FUNCTION_BLOCK PUBLIC FB_LampSetDirectDALI
VAR
	nLightLevel			: USINT;
	_nOperatingTime		: DINT;
	tonDelay			: TON;
END_VAR

IF (nLightLevel > 0) THEN
	tonDelay(IN := TRUE, PT := T#1S);
	IF (tonDelay.Q) THEN
		tonDelay(IN := FALSE);
		_nOperatingTime := _nOperatingTime + 1;
	END_IF
ELSE
	tonDelay(IN := FALSE);
END_IF

{attribute 'monitoring' := 'call'}
// Operating Time [s]
PROPERTY PUBLIC nOperatingTime : DINT
GET
nOperatingTime := _nOperatingTime;
END_GET
SET
_nOperatingTime := nOperatingTime;
END_SET
END_PROPERTY

// Sets the control value of the DALI lamp to a value between 0 and 254.
METHOD PUBLIC SetLightLevel
VAR_INPUT
	nNewLightLevel		: USINT(0..254);
END_VAR
nLightLevel := nNewLightLevel;
END_METHOD

END_FUNCTION_BLOCK

(* stored: Version 1.1.0.1, ProductVersion 3.1.4024.12
   POU FB_LampSetDirectDALI: Id {508b93c0-0778-4ff1-aedf-858d8647b6a3}, SpecialFunc None
   Property nOperatingTime: Id {62d392a4-ac0b-46a0-b328-e579ec751c57}
   Get Get: Id {329a3336-a875-4ed5-8e94-b64093512612}
   Set Set: Id {193ef73e-2d46-4bd6-be4a-aedf24d1322f}
   Method SetLightLevel: Id {fcb47fde-6ee2-43a2-b668-4bd49ce3e7e1} *)
